// TIA Portal V19 export
TYPE "M0940_HmiInterface"
   STRUCT
      PV : Real;
      SP : Real;
      EngUnitsMin : Real;
      EngUnitsMax : Real;
      P : Real;
      I : Time;
      D : Time;
      Auto_Man : Struct
         Auto : Bool;
         Manual : Bool;
         UpdateParaRec : Bool;   // Update PID Parameter Recipe depending on Loop Selection.
      END_STRUCT;
      MV : Real;   // Manual Value 0 - 100%
      OP : Real;   // PID Loop Output 0 - 100%
   END_STRUCT;
END_TYPE
